FUNCTION_BLOCK FB_LampBlinkingTest EXTENDS TcUnit.FB_TestSuite
VAR
END_VAR


//T99_test ();

METHOD PRIVATE T99_test
VAR_INST
	bJest		: BOOL;
	bKoniec		: BOOL;
END_VAR
IF (TcUnit.TEST_ORDERED ('T99_Test')) THEN
	IF (NOT bJest) THEN
		bJest					:= TRUE;
		GVL_Variable.fbLampBlinking.SetTimeOn (rIN := 100);
		GVL_Variable.fbLampBlinking.SetTimeOff (rIN := 500);
	END_IF
	GVL_Variable.fbLampBlinking.ExecuteEveryCycle_Test ();
	GVL_Variable.fbLampBlinking.ExecuteEveryCycle_Operation ();
	GVL_Variable.fbLampBlinking.ExecuteEveryCycle_Status ();
	GVL_Variable.fbLampBlinking.ExecuteEveryCycle_Error ();
	IF (bKoniec) THEN
		bJest					:= FALSE;
		TcUnit.TEST_FINISHED ();
	END_IF
END_IF
END_METHOD

END_FUNCTION_BLOCK

(* stored: Version 1.1.0.1
   POU FB_LampBlinkingTest: Id {f8af7ef6-a976-0bb5-017d-c9f286126f5d}, SpecialFunc None
   Method T99_test: Id {79133df2-cb74-013d-3ece-f01bb4f0655b} *)
